{attribute 'qualified_only'}
{attribute 'to_string'}
{attribute 'strict'}
TYPE E_INSTANCE_CMD : // instructions for fb_Instance executions
(
	NULL,
  INIT,
  DISABLE,
  ENABLE,
  WORK,
  PROCEED := 100,
  FINISH,
  CLEAR
)UINT;
END_TYPE

(* stored: Version 1.1.0.1
   DUT E_INSTANCE_CMD: Id {2ff1129e-0247-48da-b7f6-e86cac3f48a9} *)
